// TIA Portal V20 export
FUNCTION "Block_2" : Void   // FC2, LAD
{ S7_Optimized_Access := 'TRUE' }
// stored: SetENOAutomatically false
   VAR_TEMP   // added for the SCL form of the ladder/FBD networks
      _w1 : Bool;
   END_VAR
BEGIN

REGION Network 1
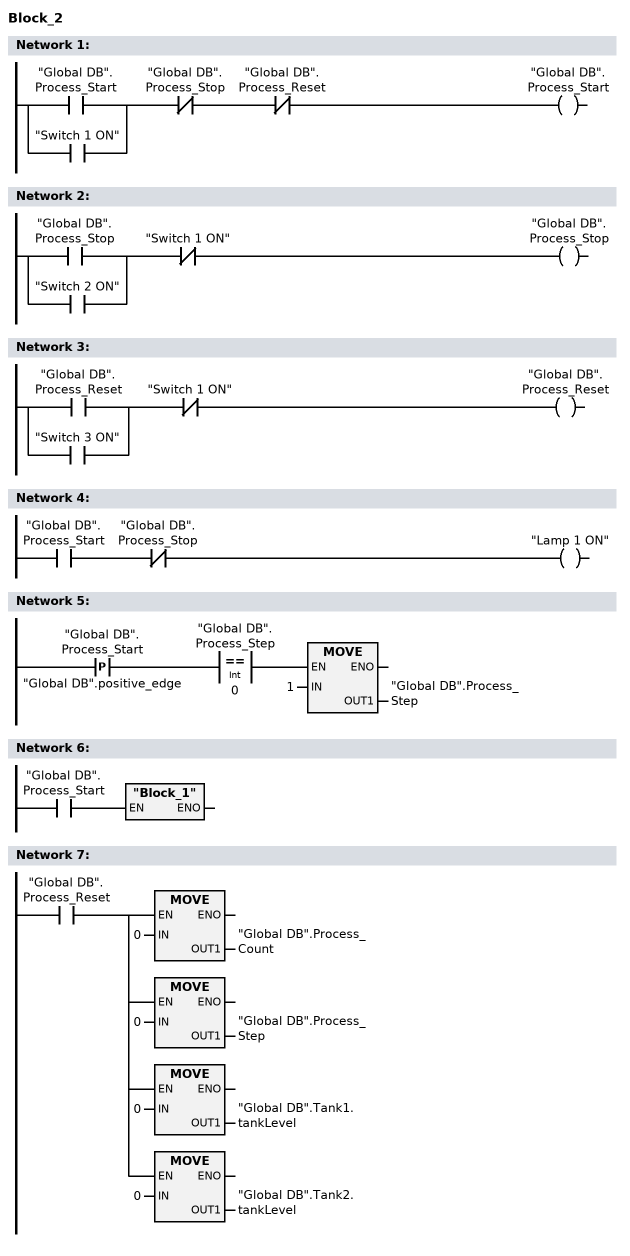
   RUNG wire#powerrail
      Contact( "Global DB".Process_Start )
      wire#w1
      I_Contact( "Global DB".Process_Stop )
      I_Contact( "Global DB".Process_Reset )
      Coil( "Global DB".Process_Start )
   END_RUNG
   RUNG wire#powerrail
      Contact( "Switch 1 ON" )
   END_RUNG wire#w1
   // the same network as SCL:
   "Global DB".Process_Start := ("Global DB".Process_Start OR "Switch 1 ON") AND NOT "Global DB".Process_Stop AND NOT "Global DB".Process_Reset;
END_REGION

REGION Network 2
   RUNG wire#powerrail
      Contact( "Global DB".Process_Stop )
      wire#w1
      I_Contact( "Switch 1 ON" )
      Coil( "Global DB".Process_Stop )
   END_RUNG
   RUNG wire#powerrail
      Contact( "Switch 2 ON" )
   END_RUNG wire#w1
   // the same network as SCL:
   "Global DB".Process_Stop := ("Global DB".Process_Stop OR "Switch 2 ON") AND NOT "Switch 1 ON";
END_REGION

REGION Network 3
   RUNG wire#powerrail
      Contact( "Global DB".Process_Reset )
      wire#w1
      I_Contact( "Switch 1 ON" )
      Coil( "Global DB".Process_Reset )
   END_RUNG
   RUNG wire#powerrail
      Contact( "Switch 3 ON" )
   END_RUNG wire#w1
   // the same network as SCL:
   "Global DB".Process_Reset := ("Global DB".Process_Reset OR "Switch 3 ON") AND NOT "Switch 1 ON";
END_REGION

REGION Network 4
   RUNG wire#powerrail
      Contact( "Global DB".Process_Start )
      I_Contact( "Global DB".Process_Stop )
      Coil( "Lamp 1 ON" )
   END_RUNG
   // the same network as SCL:
   "Lamp 1 ON" := "Global DB".Process_Start AND NOT "Global DB".Process_Stop;
END_REGION

REGION Network 5
   RUNG wire#powerrail
      P_Contact(operand := "Global DB".Process_Start, bit := "Global DB".positive_edge)
      { S7_Templates := "SrcType := Int" } EQ_Contact(in1 := "Global DB".Process_Step, in2 := 0)
      Move(in := 1, out1 => "Global DB".Process_Step)
   END_RUNG
   // the same network as SCL:
   #_w1 := "Global DB".Process_Start AND NOT "Global DB".positive_edge;   // rising edge of "Global DB".Process_Start
   "Global DB".positive_edge := "Global DB".Process_Start;
   IF #_w1 AND ("Global DB".Process_Step = 0) THEN "Global DB".Process_Step := 1; END_IF;
END_REGION

REGION Network 6
   RUNG wire#powerrail
      Contact( "Global DB".Process_Start )
      "Block_1"()
   END_RUNG
   // the same network as SCL:
   IF "Global DB".Process_Start THEN "Block_1"(); END_IF;
END_REGION

REGION Network 7
   RUNG wire#powerrail
      Contact( "Global DB".Process_Reset )
      wire#w1
      Move(in := 0, out1 => "Global DB".Process_Count)
   END_RUNG
   RUNG wire#w1
      Move(in := 0, out1 => "Global DB".Process_Step)
   END_RUNG
   RUNG wire#w1
      Move(in := 0, out1 => "Global DB".Tank1.tankLevel)
   END_RUNG
   RUNG wire#w1
      Move(in := 0, out1 => "Global DB".Tank2.tankLevel)
   END_RUNG
   // the same network as SCL:
   IF "Global DB".Process_Reset THEN
       "Global DB".Process_Count := 0;
       "Global DB".Process_Step := 0;
       "Global DB".Tank1.tankLevel := 0;
       "Global DB".Tank2.tankLevel := 0;
   END_IF;
END_REGION
END_FUNCTION
